{attribute 'qualified_only'}
{attribute 'strict'}
TYPE E_Step :
(
	(* special steps *)
	NoStep := -32767, // nessuno step    
	Unknown := -32000, // step sconosciuto
	
	(* Not Enabled or Errors*)    
	NeOrError := -990, // non abilitata o in errore
	
	(* Stop *)   
	Stop := 0, // stop
	
	
	conveyor	 :=  100	//nastro trasportare
	piston		 := 110; 		//pistone
	storage		:=120;		//magazzino	
);
END_TYPE
//  NoStep = '-32767'
//  Unknown = '-32000'
//  NeOrError = '-990'
//  conveyor = '100piston:=110; storage:=120;'

(* stored: Version 1.1.0.1, ProductVersion 3.1.4024.12
   EnumerationTextList E_Step: Id {fe3a30d3-1d96-4fc1-b1aa-f734a954498a} *)
